// TIA Portal V19 export
ORGANIZATION_BLOCK "Main"   // OB1, LAD, ProgramCycle
TITLE = "Main Program Sweep (Cycle)"
{ S7_Optimized_Access := 'TRUE' }
// stored: SetENOAutomatically false
   VAR_INPUT
      Initial_Call : Bool;   // Initial call of this OB
      Remanence : Bool;   // =True, if remanent data are available
   END_VAR
BEGIN

REGION Network 1: FC call
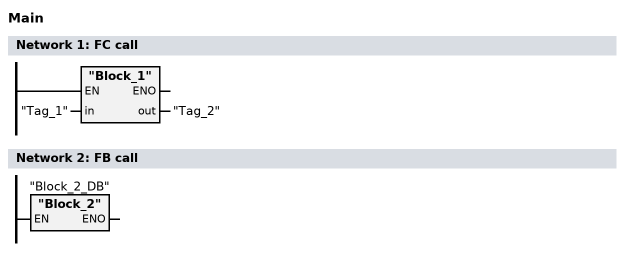
   RUNG wire#powerrail
      "Block_1"(in := "Tag_1", out => "Tag_2")
   END_RUNG
   // the same network as SCL:
   "Block_1"(in := "Tag_1", out => "Tag_2");
END_REGION

REGION Network 2: FB call
   RUNG wire#powerrail
      "Block_2_DB"()
   END_RUNG
   // the same network as SCL:
   "Block_2_DB"();   // "Block_2"
END_REGION
END_ORGANIZATION_BLOCK
